FUNCTION_BLOCK FB_Tank
VAR_INPUT
	diMixer_Running : BOOL;
	diMixer_Error : BOOL;
	diValveFill_Open : BOOL;
	diValveFill_Close : BOOL;
	diValveFill_Error : BOOL;
	diValveDrain_Open : BOOL;
	diValveDrain_Close : BOOL;
	diValveDrain_Error : BOOL;
	aiWaterLevel : WORD;
	aiWaterTemp : WORD;
	iSecImp : BOOL; //Požaduje se vstup s periodou 1 sekunda a libovolnou střídou
END_VAR

VAR_OUTPUT
	doMixer_Start : BOOL;
	doValveFill_Open : BOOL;
	doValveFill_Close : BOOL;
	doValveDrain_Open : BOOL;
	doValveDrain_Close : BOOL;
	doHeatingEnable : BOOL;
	aoReqPowerOfHeating : WORD;
END_VAR

VAR_IN_OUT
	TankData : TTank;
END_VAR

VAR
	//Konfigurace přepočtu rozsahu převodníků
	WaterTemp : TAnalogConversion := (TransducerLoLevel := 0, TransducerHiLevel := 27648, ScaledValLoLevel := 0, ScaledValHiLevel := 100);
	WaterLevel : TAnalogConversion := (TransducerLoLevel := 0, TransducerHiLevel := 27648, ScaledValLoLevel := 0, ScaledValHiLevel := 2);
	ReqOutputPower : TAnalogConversion := (ScaledValLoLevel := 0, ScaledValHiLevel := 100, TransducerLoLevel := 0, TransducerHiLevel := 27648);

	//Instance zanořených funkčních bloků
	ValveDrainCm : Valve_2DO;
	ValveFillCm : Valve_2DO;
	MixerCm : Engine_1DO;
	HeaterCm : Heater;
	FillingPhase : Filling;
	MixingPhase : Mixing;
	DrainingPhase : Draining;
	HeatingPhase : Heating;
	TON1: TON;
	RawToEng_1: RawToEng;
	RawToEng_2: RawToEng;
	EngToRaw_1: EngToRaw;
END_VAR

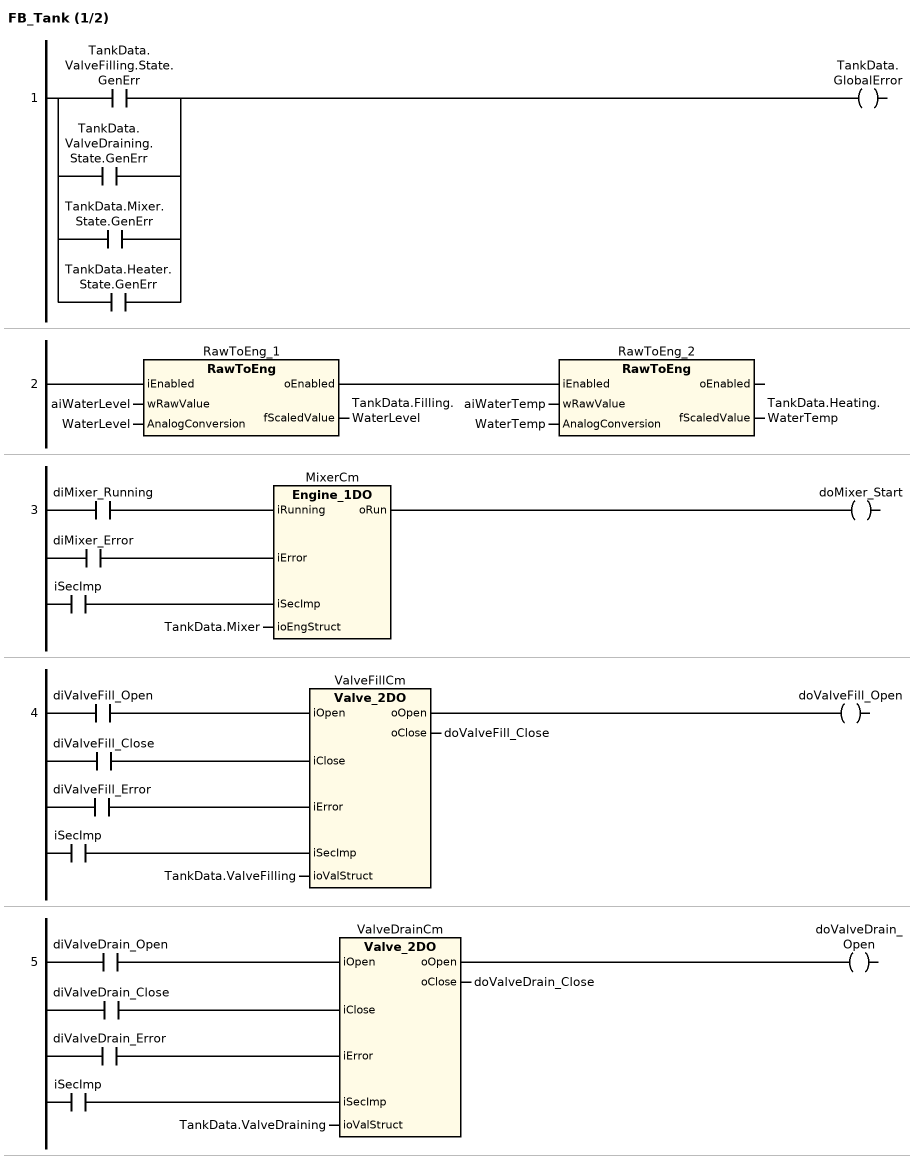
// NETWORK 1
TankData.GlobalError := TankData.ValveFilling.State.GenErr OR TankData.ValveDraining.State.GenErr OR TankData.Mixer.State.GenErr OR TankData.Heater.State.GenErr;

// NETWORK 2
RawToEng_1(
    iEnabled := TRUE,
    wRawValue := aiWaterLevel,
    AnalogConversion := WaterLevel,
    fScaledValue => TankData.Filling.WaterLevel); // RawToEng
RawToEng_2(
    iEnabled := RawToEng_1.oEnabled,
    wRawValue := aiWaterTemp,
    AnalogConversion := WaterTemp,
    fScaledValue => TankData.Heating.WaterTemp); // RawToEng

// NETWORK 3
MixerCm(
    iRunning := diMixer_Running,
    iError := diMixer_Error,
    iSecImp := iSecImp,
    ioEngStruct := TankData.Mixer); // Engine_1DO
doMixer_Start := MixerCm.oRun;

// NETWORK 4
ValveFillCm(
    iOpen := diValveFill_Open,
    iClose := diValveFill_Close,
    iError := diValveFill_Error,
    iSecImp := iSecImp,
    ioValStruct := TankData.ValveFilling,
    oClose => doValveFill_Close); // Valve_2DO
doValveFill_Open := ValveFillCm.oOpen;

// NETWORK 5
ValveDrainCm(
    iOpen := diValveDrain_Open,
    iClose := diValveDrain_Close,
    iError := diValveDrain_Error,
    iSecImp := iSecImp,
    ioValStruct := TankData.ValveDraining,
    oClose => doValveDrain_Close); // Valve_2DO
doValveDrain_Open := ValveDrainCm.oOpen;

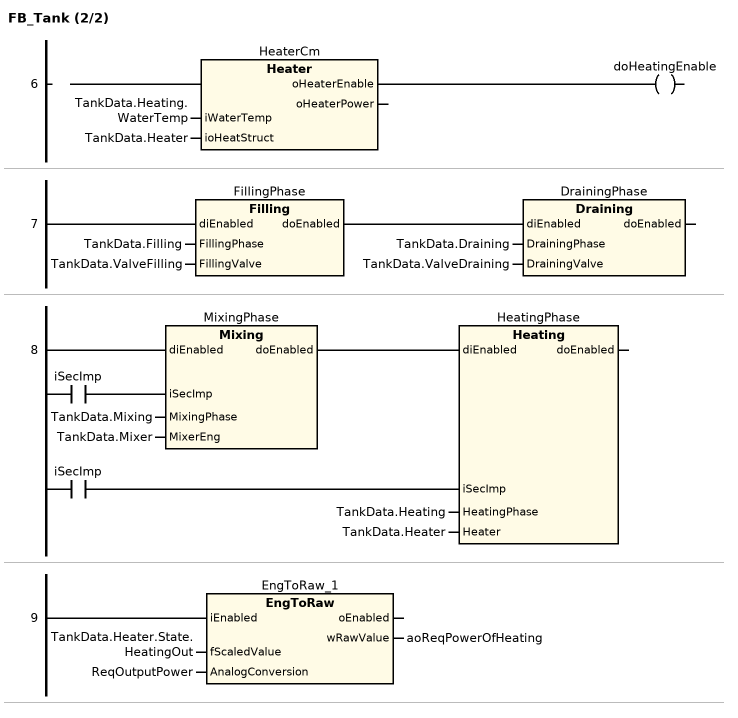
// NETWORK 6
HeaterCm(iWaterTemp := TankData.Heating.WaterTemp, ioHeatStruct := TankData.Heater); // Heater
doHeatingEnable := HeaterCm.oHeaterEnable;

// NETWORK 7
FillingPhase(diEnabled := TRUE, FillingPhase := TankData.Filling, FillingValve := TankData.ValveFilling); // Filling
DrainingPhase(
    diEnabled := FillingPhase.doEnabled,
    DrainingPhase := TankData.Draining,
    DrainingValve := TankData.ValveDraining); // Draining

// NETWORK 8
MixingPhase(
    diEnabled := TRUE,
    iSecImp := iSecImp,
    MixingPhase := TankData.Mixing,
    MixerEng := TankData.Mixer); // Mixing
HeatingPhase(
    diEnabled := MixingPhase.doEnabled,
    iSecImp := iSecImp,
    HeatingPhase := TankData.Heating,
    Heater := TankData.Heater); // Heating

// NETWORK 9
EngToRaw_1(
    iEnabled := TRUE,
    fScaledValue := TankData.Heater.State.HeatingOut,
    AnalogConversion := ReqOutputPower,
    wRawValue => aoReqPowerOfHeating); // EngToRaw

END_FUNCTION_BLOCK

(* stored: Version 1.1.0.1, ProductVersion 3.1.4024.13
   POU FB_Tank: Id {c85dc8a0-9f5f-473b-9759-baf364dbe5e8}, SpecialFunc None *)
